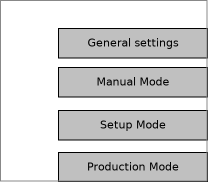
VISUALIZATION MainWindow  // 208x182
    Rectangle (58,152 150x30), "Production Mode", tooltip "Operation mode supposed to be used for production with slightly reduced measurement frequency."
        OnMouseClick: change screen: Production_Mode
    Rectangle (58,110 150x30), "Setup Mode", tooltip "Operation mode with increased measuring frequency in order to fine tune the process (e.g. reference values) according to your needs."
        OnMouseClick: change screen: Setup_Mode
    Rectangle (58,67 150x30), "Manual Mode", tooltip "Allows manual control (start/stop) of each and every subsystem."
        OnMouseClick: change screen: Manual_Mode
    Rectangle (58,28 150x30), "General settings", tooltip "Allows to adjust general system parameters, which will be applied in all different modes of operation."
        OnMouseClick: change screen: GeneralSettings
END_VISUALIZATION

(* stored: Version 1.1.0.1
   Visu MainWindow: Id {d82e5b75-be32-4ecc-898d-7f43aa342158} *)
